(* CODESYS project InstalacaoPortuaria.project

Project tree, tasks and I/O mapping:
  Device : CODESYS Control Win V3, 3S - Smart Software Solutions GmbH, order no. 305021, version 3.5.11.40
    application Application
      libraries: Standard, * (System)
      task MainTask (cyclic, interval t#20ms, priority 0) calls PLC_PRG
      task Simulacao (cyclic, interval t#500ms, priority 1) calls SIMULACAO
      program PLC_PRG [SFC]: _aDESCARREGAMENTO_active, _aCARREGAMENTO_active, _aALARMES_active, _aS5_entry, _aSC2_entry, _aSC3_entry, _aSC4_entry, _aSC5_entry, _aSC6_entry, _aSC7_entry, _aS7_active, _aSC10_active, _aS1_active, _aSC2_active, _aSELECAO_DESC_active, _aSELECAO_CARR_active, _aInit_active, _aS3_active
      program SIMULACAO [SFC]: _aSCARREGAMENTO_active, _aSDESCARREGAMENTO_active, _aSD2_active, _aSD3_entry, _aSC2_active, _aSSILO_active, _aSC3_entry, _aSD1_entry, _aSC0_entry, _aSC0_exit, _aSC3_exit, _aSD0_entry, _aSD0_exit, _aSD3_exit
      Symbols
*)

// Device/Application/PLC_PRG
PROGRAM PLC_PRG
VAR_INPUT
	// VAGAO GRANELEIRO
	// VARIAVEL REFERENTE AO SENSOR DE POSICIONAMENTO DO VAGAO GRANELEIRO
	VAGAO: BOOL:= 0;
	// QUANTIDADE DE GRAOS NO VAGAO GANELEIRO
	GRAOS: REAL:=0;
	
	// TRANSPORTADOR DE ENTRADA
	// CELULA DE CARGA DO TRANSPORTADOR
	C_TR_01: BOOL:= 0;
	
	// SILOS DE ARMAZENAGEM
	// CELULAS DE CARGA
	C_AS_01: REAL:= 0;	
	C_AS_02: REAL:= 0;
	// CHAVE DE BAIXO NIVEL
	L_AS_01: BOOL:= 0;
	L_AS_02: BOOL:= 0;
	// CHAVE DE ALTO NIVEL
	H_AS_01: BOOL:= 0;
	H_AS_02: BOOL:= 0;
	
	// ALIMENTADORES DA MOEGA 
	// INDICADOR DE GRAOS
	C_AL_01: BOOL:= 0;
	C_AL_02: BOOL:= 0;
	
	// MOEGA
	// CONTABILIZA O PESO DOS GRAOS TRANSFERIDOS
	C_MO_01: REAL:= 0;
	
	// TRANSPORTADOR DE SAIDA
	// CELULA DE CARGA DO TRANSPORTADOR
	C_TR_02: BOOL:= 0;
	
	// ALIMENTADOR DE SAIDA
	// SENSOR CAMINHAO CORRETAMENTE POSICIONADO
	CAMINHAO: BOOL:= 0;
	
	// SENSORES DE CHEGADA
	// CHEGADA VAGAO
	VAGAO_C: BOOL:= 0;
	// CHEGADA CAMINHAO
	CAMINHAO_C: BOOL:= 0;
	
	// SENSORES DE SAIDA
	// SAIDA VAGAO
	VAGAO_S: BOOL:= 0;
	// SAIDA CAMINHAO
	CAMINHAO_S: BOOL:= 0;

END_VAR
VAR
	// MODO CARREGAMENTO
	SELEC_CARR_MAN: BOOL:= 0;
	CARR_MAN: BOOL:= 0;
	// INICIA CARREGAMENTO AUTOMATICO
	CARREGAR: BOOL:= 0;
	// CARREGAMENTO NÃO PODE SER ACIONADO
	I_NOT_CARR: BOOL:= 0;
	// ALARME GRAOS INSUFICIENTES
	I_GRAOS: BOOL:= 0;
	// MODO DESCARREGAMENTO
	SELEC_DESC_MAN: BOOL:= 0;
	DESC_MAN: BOOL:= 0;
	// DESCARREGAMENTO NÃO PODE SER ACIONADO
	I_NOT_DESC: BOOL:= 0;
	// INICIA DESCARREGAMENTO AUTOMATICO
	DESCARREGAR: BOOL:= 0;		

	// VARIAVEIS DE INTERFACE
	//VAGAO GRANELEIRO
	// SENSOR DE POSICIONAMENTO DO VAGAO GRANELEIRO
	I_VAGAO: BOOL:= 0;
	
	//TRANSPORTADOR DE ENTRADA
	// ESTADO DO TRANSPORTADOR DE ENTRADA
	I_TR_01: BOOL:= 0;
	// CELULA DE CARGA DO TRANSPORTADOR
	I_C_TR_01: BOOL:= 0;
	// INDICACAO QUE O TRANSPORTADOR ESTÁ LIGADO E VAZIO POR MAIS DE 5S
	I_VAZIO_TR_01: BOOL:= 0;
	
	// DESVIADOR DE MANGUEIRA
	I_MG_01: BOOL:= 0;
	
	// SILOS DE ARMAZENAGEM
	// CELULAS DE CARGA
	I_C_AS_01: REAL:= 0;	
	I_C_AS_02: REAL:= 0;
	// CHAVE DE BAIXO NIVEL
	I_L_AS_01: BOOL:= 0;
	I_L_AS_02: BOOL:= 0;
	// CHAVE DE ALTO NIVEL
	I_H_AS_01: BOOL:= 0;
	I_H_AS_02: BOOL:= 0;
	// SISTEMA DE VENTILACAO
	I_V_AS_01: BOOL:= 0;
	I_V_AS_02: BOOL:= 0;
	
	// ALIMENTADORES DA MOEGA 
	I_AL_01: BOOL:= 0;
	I_AL_02: BOOL:= 0;
	// ALARME LIGADO E VAZIO POR MAIS DE 5S
	I_VAZIO_AL_01: BOOL:= 0;
	I_VAZIO_AL_02: BOOL:= 0;
	// INDICADOR DE GRAOS
	I_C_AL_01: BOOL:= 0;
	I_C_AL_02: BOOL:= 0;
	
	// MOEGA
	// ESTADO DA MOEGA
	I_MO_01: BOOL:= 0;
	// CONTABILIZA O PESO DOS GRAOS TRANSFERIDOS
	I_C_MO_01: REAL:= 0;
	// ALARME TRANSPORTADOR DESLIGADO E PESO DIFERENTE DE 0
	I_CHEIO_MO_01: BOOL:= 0; 
	
	//TRANSPORTADOR DE SAIDA
	// ESTADO DO TRANSPORTADOR DE SAIDA
	I_TR_02: BOOL:= 0;
	// CELULA DE CARGA DO TRANSPORTADOR
	I_C_TR_02: BOOL:= 0;
	// INDICACAO QUE O TRANSPORTADOR ESTÁ LIGADO E VAZIO POR MAIS DE 5S
	I_VAZIO_TR_02: BOOL:= 0;
	// INDICACAO QUE O TRANSPORTADOR ESTÁ LIGADO E ALIMENTADOR DESLIGADO
	I_LIGADO_TR_02: BOOL:= 0;
	
	// ALIMENTADOR DE SAIDA
	// ESTADO DO ALIMENTADOR DE SAIDA
	I_AL_03: BOOL:= 0;
	// SENSOR CAMINHAO CORRETAMENTE POSICIONADO
	I_CAMIHAO: BOOL:= 0;
	// ALARME ALIMENTADOR LIGADO CAMINHAO DESCONECTADO
	I_LIGADO_AL_03: BOOL:=0;
	
	// CAPACIDADE DO CAMINHAO
	I_CAPACIDADE: REAL:= 0;
	
	// SENSORES DE CHEGADA
	// CHEGADA VAGAO
	I_VAGAO_C: BOOL:= 0;
	// CHEGADA CAMINHAO
	I_CAMINHAO_C: BOOL:= 0;
	
	// SENSORES DE SAIDA
	// SAIDA VAGAO
	I_VAGAO_S: BOOL:= 0;
	// SAIDA CAMINHAO
	I_CAMINHAO_S: BOOL:= 0;
	
	TON_0: TON;
	TON_1: TON;
END_VAR
VAR_OUTPUT
	
	//TRANSPORTADOR DE ENTRADA
	// ACIONA O TRANSPORTADOR DE ENTRADA
	TR_01: BOOL:= 0;

	//DESVIADOR DE MANGUEIRA
	MG_01: BOOL:= 0;

	// SILOS DE ARMAZENAGEM
	// SISTEMA DE VENTILACAO
	V_AS_01: BOOL:= 0;
	V_AS_02: BOOL:= 0;
	
	//ALIMENTADORES DA MOEGA 
	AL_01: BOOL:= 0;
	AL_02: BOOL:= 0;
	
	// MOEGA
	// ESTADO DA MOEGA
	MO_01: BOOL:= 0;
	
	//TRANSPORTADOR DE SAIDA
	// ESTADO DO TRANSPORTADOR DE SAIDA
	TR_02: BOOL:= 0;
	
	// ALIMENTADOR DE SAIDA
	// ESTADO DO ALIMENTADOR DE SAIDA
	AL_03: BOOL:= 0;

END_VAR

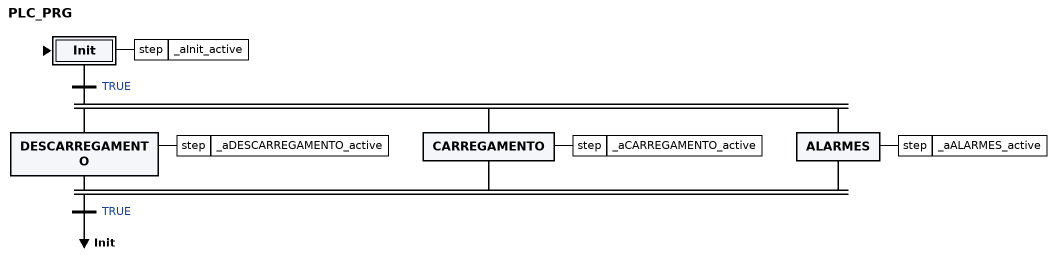
INITIAL_STEP Init:
    _aInit_active(N);  // step action
END_STEP
TRANSITION FROM Init TO (DESCARREGAMENTO, CARREGAMENTO, ALARMES)
    := TRUE;
END_TRANSITION
STEP DESCARREGAMENTO:
    _aDESCARREGAMENTO_active(N);  // step action
END_STEP
STEP CARREGAMENTO:
    _aCARREGAMENTO_active(N);  // step action
END_STEP
STEP ALARMES:
    _aALARMES_active(N);  // step action
END_STEP
TRANSITION FROM (DESCARREGAMENTO, CARREGAMENTO, ALARMES) TO Init
    := TRUE;
END_TRANSITION

ACTION _aDESCARREGAMENTO_active:
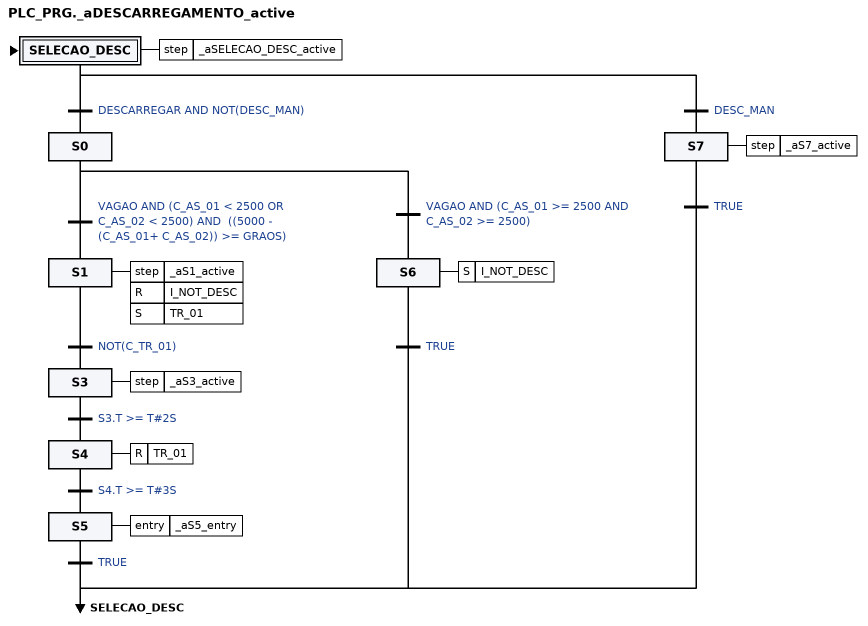
INITIAL_STEP SELECAO_DESC:
    _aSELECAO_DESC_active(N);  // step action
END_STEP
TRANSITION FROM SELECAO_DESC TO S0
    := DESCARREGAR AND NOT(DESC_MAN);
END_TRANSITION
STEP S0:
END_STEP
TRANSITION FROM S0 TO S1
    := VAGAO AND (C_AS_01 < 2500 OR C_AS_02 < 2500) AND ((5000 - (C_AS_01+ C_AS_02)) >= GRAOS);
END_TRANSITION
STEP S1:
    _aS1_active(N);  // step action
    I_NOT_DESC(R);
    TR_01(S);
END_STEP
TRANSITION FROM S1 TO S3
    := NOT(C_TR_01);
END_TRANSITION
STEP S3:
    _aS3_active(N);  // step action
END_STEP
TRANSITION FROM S3 TO S4
    := S3.T >= T#2S;
END_TRANSITION
STEP S4:
    TR_01(R);
END_STEP
TRANSITION FROM S4 TO S5
    := S4.T >= T#3S;
END_TRANSITION
STEP S5:
    _aS5_entry(P1);  // entry action
END_STEP
TRANSITION FROM S5 TO SELECAO_DESC
    := TRUE;
END_TRANSITION
TRANSITION FROM S0 TO S6
    := VAGAO AND (C_AS_01 >= 2500 AND C_AS_02 >= 2500);
END_TRANSITION
STEP S6:
    I_NOT_DESC(S);
END_STEP
TRANSITION FROM S6 TO SELECAO_DESC
    := TRUE;
END_TRANSITION
TRANSITION FROM SELECAO_DESC TO S7
    := DESC_MAN;
END_TRANSITION
STEP S7:
    _aS7_active(N);  // step action
END_STEP
TRANSITION FROM S7 TO SELECAO_DESC
    := TRUE;
END_TRANSITION
// branch label Branch2__aDESCARREGAMENTO_entry
END_ACTION

ACTION _aCARREGAMENTO_active:
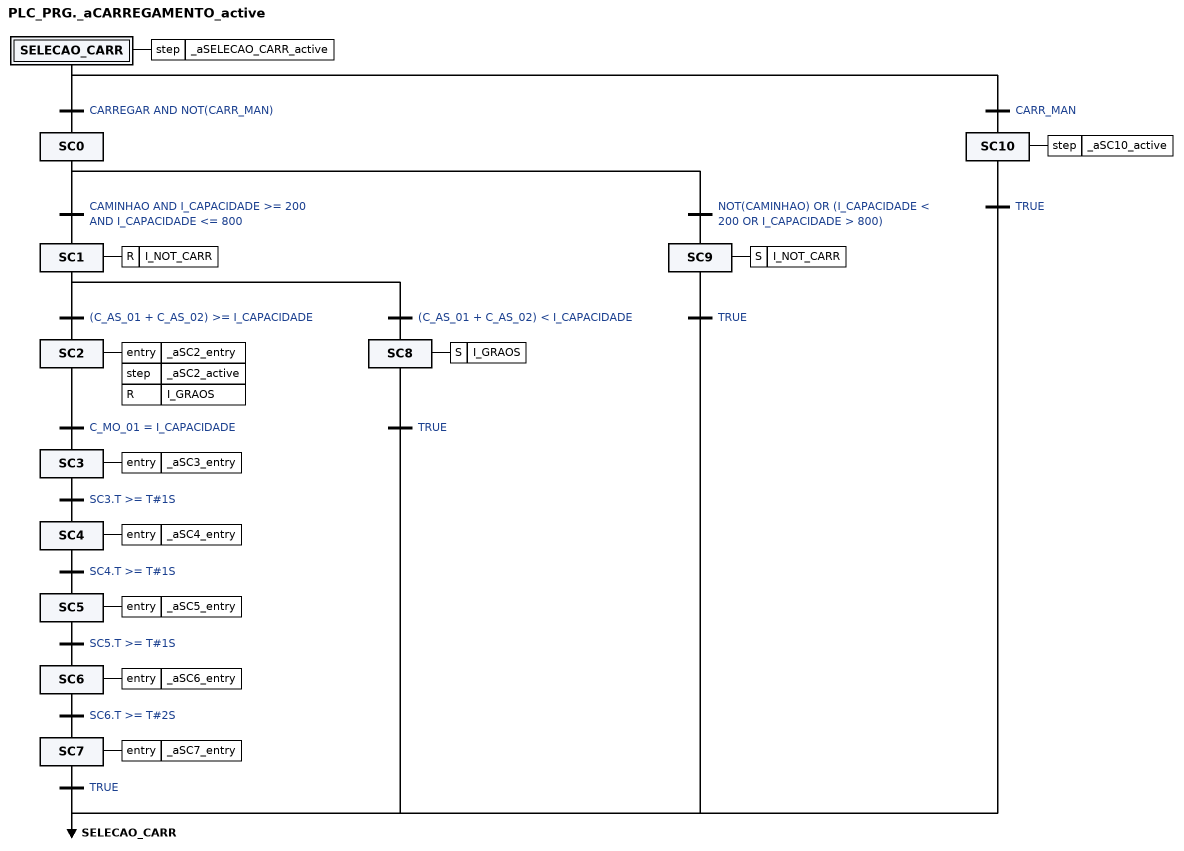
INITIAL_STEP _SELECAO_CARR:  // name as stored:  SELECAO_CARR
    _aSELECAO_CARR_active(N);  // step action
END_STEP
TRANSITION FROM _SELECAO_CARR TO SC0
    := CARREGAR AND NOT(CARR_MAN);
END_TRANSITION
STEP SC0:
END_STEP
TRANSITION FROM SC0 TO SC1
    := CAMINHAO AND I_CAPACIDADE >= 200 AND I_CAPACIDADE <= 800;
END_TRANSITION
STEP SC1:
    I_NOT_CARR(R);
END_STEP
TRANSITION FROM SC1 TO SC2
    := (C_AS_01 + C_AS_02) >= I_CAPACIDADE;
END_TRANSITION
STEP SC2:
    _aSC2_entry(P1);  // entry action
    _aSC2_active(N);  // step action
    I_GRAOS(R);
END_STEP
TRANSITION FROM SC2 TO SC3
    := C_MO_01 = I_CAPACIDADE;
END_TRANSITION
STEP SC3:
    _aSC3_entry(P1);  // entry action
END_STEP
TRANSITION FROM SC3 TO SC4
    := SC3.T >= T#1S;
END_TRANSITION
STEP SC4:
    _aSC4_entry(P1);  // entry action
END_STEP
TRANSITION FROM SC4 TO SC5
    := SC4.T >= T#1S;
END_TRANSITION
STEP SC5:
    _aSC5_entry(P1);  // entry action
END_STEP
TRANSITION FROM SC5 TO SC6
    := SC5.T >= T#1S;
END_TRANSITION
STEP SC6:
    _aSC6_entry(P1);  // entry action
END_STEP
TRANSITION FROM SC6 TO SC7
    := SC6.T >= T#2S;
END_TRANSITION
STEP SC7:
    _aSC7_entry(P1);  // entry action
END_STEP
TRANSITION FROM SC7 TO SELECAO_CARR
    := TRUE;
END_TRANSITION
TRANSITION FROM SC1 TO SC8
    := (C_AS_01 + C_AS_02) < I_CAPACIDADE;
END_TRANSITION
STEP SC8:
    I_GRAOS(S);
END_STEP
TRANSITION FROM SC8 TO SELECAO_CARR
    := TRUE;
END_TRANSITION
TRANSITION FROM SC0 TO SC9
    := NOT(CAMINHAO) OR (I_CAPACIDADE < 200 OR I_CAPACIDADE > 800);
END_TRANSITION
STEP SC9:
    I_NOT_CARR(S);
END_STEP
TRANSITION FROM SC9 TO SELECAO_CARR
    := TRUE;
END_TRANSITION
TRANSITION FROM _SELECAO_CARR TO SC10
    := CARR_MAN;
END_TRANSITION
STEP SC10:
    _aSC10_active(N);  // step action
END_STEP
TRANSITION FROM SC10 TO SELECAO_CARR
    := TRUE;
END_TRANSITION
// branch label Branch2__aCARREGAMENTO_active
// branch label Branch1__aCARREGAMENTO_active
// branch label Branch0__aCARREGAMENTO_active
END_ACTION

ACTION _aALARMES_active:
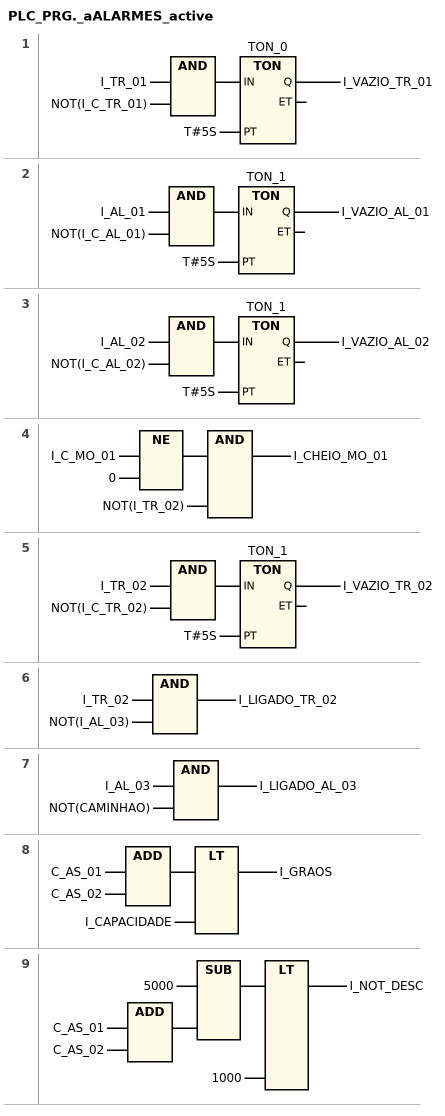
// NETWORK 1
TON_0(IN := I_TR_01 AND (NOT(I_C_TR_01)), PT := T#5S); // TON
I_VAZIO_TR_01 := TON_0.Q;

// NETWORK 2
TON_1(IN := I_AL_01 AND (NOT(I_C_AL_01)), PT := T#5S); // TON
I_VAZIO_AL_01 := TON_1.Q;

// NETWORK 3
TON_1(IN := I_AL_02 AND (NOT(I_C_AL_02)), PT := T#5S); // TON
I_VAZIO_AL_02 := TON_1.Q;

// NETWORK 4
I_CHEIO_MO_01 := I_C_MO_01 <> 0 AND (NOT(I_TR_02));

// NETWORK 5
TON_1(IN := I_TR_02 AND (NOT(I_C_TR_02)), PT := T#5S); // TON
I_VAZIO_TR_02 := TON_1.Q;

// NETWORK 6
I_LIGADO_TR_02 := I_TR_02 AND (NOT(I_AL_03));

// NETWORK 7
I_LIGADO_AL_03 := I_AL_03 AND (NOT(CAMINHAO));

// NETWORK 8
I_GRAOS := C_AS_01 + C_AS_02 < I_CAPACIDADE;

// NETWORK 9
I_NOT_DESC := 5000 - (C_AS_01 + C_AS_02) < 1000;
END_ACTION

ACTION _aS5_entry:
IF (I_V_AS_01 = 1) THEN
	V_AS_01:= 0;
END_IF
IF (I_V_AS_02 = 1) THEN
	V_AS_02:= 0;
END_IF
I_V_AS_01:= V_AS_01;
I_V_AS_02:= V_AS_02;
END_ACTION

ACTION _aSC2_entry:
//ALIMENTADOR DE SAÍDA
AL_03 := 1;
I_AL_03 := AL_03;
//TRANSPORTADOR DE SAÍDA
TR_02 := 1;
I_TR_02 := TR_02;
//MOEGA
MO_01 := 1;
I_MO_01 := MO_01;
END_ACTION

ACTION _aSC3_entry:
//SILO
IF (I_AL_01 = 1) THEN
	AL_01 := 0;
END_IF
IF (I_AL_02 = 1) THEN
	AL_02 := 0;
END_IF
I_AL_01 := AL_01;
I_AL_02 := AL_02;
END_ACTION

ACTION _aSC4_entry:
//MOEGA
MO_01 := 0;
I_MO_01 := MO_01;
END_ACTION

ACTION _aSC5_entry:
//TRANSPORTADOR DE SAÍDA
TR_02 := 0;
I_TR_02 := TR_02;
END_ACTION

ACTION _aSC6_entry:
//ALIMENTADOR DE SAÍDA
AL_03 := 0;
I_AL_03 := AL_03;
END_ACTION

ACTION _aSC7_entry:
//SILO
IF (I_V_AS_01 = 1) THEN
	V_AS_01 := 0;
END_IF
IF (I_V_AS_02 = 1) THEN
	V_AS_02 := 0;
END_IF
I_V_AS_01 := V_AS_01;
I_V_AS_02 := V_AS_02;
END_ACTION

ACTION _aS7_active:
// TRANSPORTADOR DE ENTRADA
IF(I_TR_01 = 1)THEN
	TR_01:= 1;
ELSE
	TR_01:= 0;
END_IF
// DESVIADOR DA MANGUEIRA
IF(I_MG_01 = 1)THEN
	MG_01:= 1;
ELSE
	MG_01:= 0;
END_IF
// SILO DE ARMAZENAGEM 1
IF(I_V_AS_01 = 1)THEN
	V_AS_01:= 1;
ELSE
	V_AS_01:= 0;
END_IF
// SILO DE ARMAZENAGEM 2
IF(I_V_AS_02 = 1)THEN
	V_AS_02:= 1;
ELSE
	V_AS_02:= 0;
END_IF
END_ACTION

ACTION _aSC10_active:
// SILO DE ARMAZENAGEM 1
IF(I_V_AS_01 = 1)THEN
	V_AS_01:= 1;
ELSE
	V_AS_01:= 0;
END_IF
// SILO DE ARMAZENAGEM 2
IF(I_V_AS_02 = 1)THEN
	V_AS_02:= 1;
ELSE
	V_AS_02:= 0;
END_IF
// ALIMENTADOR DA MOEGA 1
IF(I_AL_01 = 1)THEN
	AL_01:= 1;
ELSE
	AL_01:= 0;
END_IF
// ALIMENTADOR DA MOEGA 2
IF(I_AL_02 = 1)THEN
	AL_02:= 1;
ELSE
	AL_02:= 0;
END_IF
// MOEGA
IF(I_MO_01 = 1)THEN
	MO_01:= 1;
ELSE
	MO_01:= 0;
END_IF
// TRANSPORTADOR DE SAÍDA
IF(I_TR_02 = 1)THEN
	TR_02:= 1;
ELSE
	TR_02:= 0;
END_IF
// ALIMENTADOR DE SAÍDA
IF(I_AL_03 = 1)THEN
	AL_03:= 1;
ELSE
	AL_03:= 0;
END_IF
END_ACTION

ACTION _aS1_active:
IF (C_AS_01 <= C_AS_02) THEN
		MG_01:= 0;
ELSE
		MG_01:= 1;
END_IF
I_MG_01:= MG_01;
I_C_AS_01:= C_AS_01; 
I_C_AS_02:= C_AS_02;

IF (I_MG_01 = 0) THEN
	V_AS_01:= 1;
ELSE
	V_AS_02:= 1;
END_IF
I_V_AS_01:= V_AS_01;
I_V_AS_02:= V_AS_02;
END_ACTION

ACTION _aSC2_active:
//SILO
IF (C_AS_01 >= C_AS_02) THEN
		AL_01 := 1;
		AL_02 := 0;
		V_AS_01 := 1;
		V_AS_02 := 0;
ELSE
		AL_01 := 0;
		AL_02 := 1;
		V_AS_01 := 0;
		V_AS_02 := 1;
END_IF
I_AL_01 := AL_01;
I_AL_02 := AL_02;
I_V_AS_01 := V_AS_01;
I_V_AS_02 := V_AS_02;

I_C_AS_01:= C_AS_01; 
I_C_AS_02:= C_AS_02;
END_ACTION

ACTION _aSELECAO_DESC_active:
IF (TR_01 = 0) AND (I_VAZIO_TR_01 = 0) THEN
	DESC_MAN:= SELEC_DESC_MAN;
END_IF
END_ACTION

ACTION _aSELECAO_CARR_active:
IF (AL_01 = 0) AND (AL_02 = 0) AND (AL_03 = 0) AND (MO_01 = 0) AND (TR_02 = 0) 
AND (I_VAZIO_AL_01 = 0) AND (I_VAZIO_AL_02 = 0) AND (I_CHEIO_MO_01 = 0) 
AND (I_VAZIO_TR_02 = 0) AND (I_LIGADO_TR_02 = 0) AND (I_LIGADO_AL_03 = 0)
AND (I_GRAOS = 0) THEN
	CARR_MAN:= SELEC_CARR_MAN;
END_IF
END_ACTION

ACTION _aInit_active:
//CHAVES DE BAIXO NÍVEL
I_L_AS_01:= L_AS_01;
I_L_AS_02:= L_AS_02;
//CHAVES DE ALTO NÍVEL
I_H_AS_01:= H_AS_01;
I_H_AS_02:= H_AS_02;
//SENSORES DE CHEGADA
I_CAMINHAO_C:= CAMINHAO_C;
I_VAGAO_C:= VAGAO_C;
//SENSORES DE SAIDA
I_CAMINHAO_S:= CAMINHAO_S;
I_VAGAO_S:= VAGAO_S;
//SENSOR VAGAO POSICIONADO
I_VAGAO:= VAGAO;
END_ACTION

ACTION _aS3_active:
I_C_AS_01:= C_AS_01; 
I_C_AS_02:= C_AS_02;
END_ACTION

END_PROGRAM

// Device/Application/SIMULACAO
PROGRAM SIMULACAO

VAR
	T1: TON;
	T2: TON;
	GRAOS_VAGAO: REAL := 0;
END_VAR

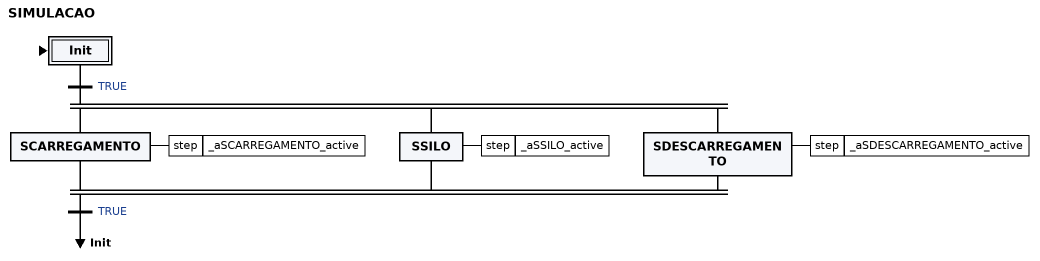
INITIAL_STEP Init:
END_STEP
TRANSITION FROM Init TO (SCARREGAMENTO, SSILO, SDESCARREGAMENTO)
    := TRUE;
END_TRANSITION
STEP SCARREGAMENTO:
    _aSCARREGAMENTO_active(N);  // step action
END_STEP
STEP SSILO:
    _aSSILO_active(N);  // step action
END_STEP
STEP SDESCARREGAMENTO:
    _aSDESCARREGAMENTO_active(N);  // step action
END_STEP
TRANSITION FROM (SCARREGAMENTO, SSILO, SDESCARREGAMENTO) TO Init
    := TRUE;
END_TRANSITION

ACTION _aSCARREGAMENTO_active:
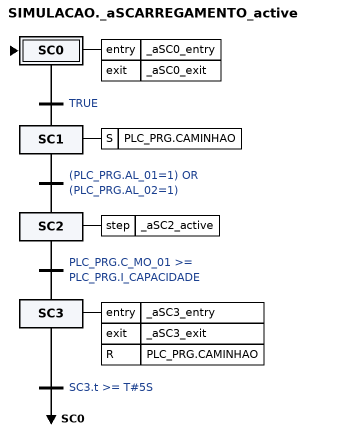
INITIAL_STEP SC0:
    _aSC0_entry(P1);  // entry action
    _aSC0_exit(P0);  // exit action
END_STEP
TRANSITION FROM SC0 TO SC1
    := TRUE;
END_TRANSITION
STEP SC1:
    PLC_PRG.CAMINHAO(S);
END_STEP
TRANSITION FROM SC1 TO SC2
    := (PLC_PRG.AL_01=1) OR (PLC_PRG.AL_02=1);
END_TRANSITION
STEP SC2:
    _aSC2_active(N);  // step action
END_STEP
TRANSITION FROM SC2 TO SC3
    := PLC_PRG.C_MO_01 >= PLC_PRG.I_CAPACIDADE;
END_TRANSITION
STEP SC3:
    _aSC3_entry(P1);  // entry action
    _aSC3_exit(P0);  // exit action
    PLC_PRG.CAMINHAO(R);
END_STEP
TRANSITION FROM SC3 TO SC0
    := SC3.t >= T#5S;
END_TRANSITION
END_ACTION

ACTION _aSDESCARREGAMENTO_active:
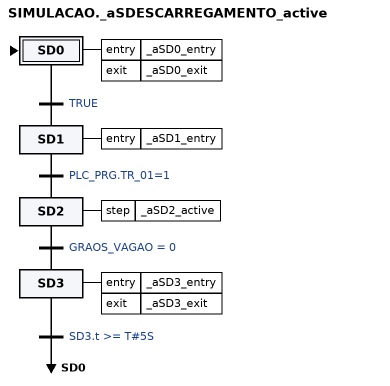
INITIAL_STEP SD0:
    _aSD0_entry(P1);  // entry action
    _aSD0_exit(P0);  // exit action
END_STEP
TRANSITION FROM SD0 TO SD1
    := TRUE;
END_TRANSITION
STEP SD1:
    _aSD1_entry(P1);  // entry action
END_STEP
TRANSITION FROM SD1 TO SD2
    := PLC_PRG.TR_01=1;
END_TRANSITION
STEP SD2:
    _aSD2_active(N);  // step action
END_STEP
TRANSITION FROM SD2 TO SD3
    := GRAOS_VAGAO = 0;
END_TRANSITION
STEP SD3:
    _aSD3_entry(P1);  // entry action
    _aSD3_exit(P0);  // exit action
END_STEP
TRANSITION FROM SD3 TO SD0
    := SD3.t >= T#5S;
END_TRANSITION
END_ACTION

ACTION _aSD2_active:
PLC_PRG.C_TR_01:= 1;
T1(IN:=TRUE,PT:=T#1S);
IF(T1.Q = 1)THEN
	IF (PLC_PRG.MG_01 = 0) THEN
		GRAOS_VAGAO:= GRAOS_VAGAO - 100;
		PLC_PRG.GRAOS:= GRAOS_VAGAO;
		PLC_PRG.C_AS_01:= PLC_PRG.C_AS_01+100;
	ELSE
		GRAOS_VAGAO:= GRAOS_VAGAO - 100;
		PLC_PRG.GRAOS:= GRAOS_VAGAO;
		PLC_PRG.C_AS_02:= PLC_PRG.C_AS_02+100;
	END_IF
	T1(IN:=FALSE);
END_IF
END_ACTION

ACTION _aSD3_entry:
PLC_PRG.C_TR_01:= 0;
PLC_PRG.VAGAO:= 0;
PLC_PRG.VAGAO_S:= 1;
END_ACTION

ACTION _aSC2_active:
PLC_PRG.C_TR_02:= 1;
T2(IN:=TRUE,PT:=T#1S);
IF(T2.Q = 1)THEN
	IF (PLC_PRG.AL_01 = 1) THEN
		IF (PLC_PRG.C_AS_01>=50) THEN
			PLC_PRG.C_AL_01:= 1;
			PLC_PRG.C_AS_01:= PLC_PRG.C_AS_01 - 50;
			PLC_PRG.C_MO_01:= PLC_PRG.C_MO_01 + 50;
		END_IF
	END_IF
	IF (PLC_PRG.AL_02 = 1) THEN
		IF (PLC_PRG.C_AS_02>=50) THEN
			PLC_PRG.C_AL_02:= 1;
			PLC_PRG.C_AS_02:= PLC_PRG.C_AS_02 - 50;
			PLC_PRG.C_MO_01:= PLC_PRG.C_MO_01 + 50;
		END_IF
	END_IF
	T2(IN:=FALSE);
END_IF
END_ACTION

ACTION _aSSILO_active:
//SIMULAÇÃO DAS CHAVES DE ALTO E BAIXO NÍVEL DOS SILOS

IF (PLC_PRG.C_AS_01<=100) THEN
	PLC_PRG.L_AS_01:= 1;
ELSIF (PLC_PRG.C_AS_01>=2400) THEN
	PLC_PRG.H_AS_01:= 1;
ELSE 
	PLC_PRG.L_AS_01:= 0;
	PLC_PRG.H_AS_01:= 0;
END_IF

IF (PLC_PRG.C_AS_02<=100) THEN
	PLC_PRG.L_AS_02:= 1;
ELSIF (PLC_PRG.C_AS_02>=2400) THEN
	PLC_PRG.H_AS_02:= 1;
ELSE 
	PLC_PRG.L_AS_02:= 0;
	PLC_PRG.H_AS_02:= 0;
END_IF
END_ACTION

ACTION _aSC3_entry:
PLC_PRG.C_TR_02:= 0;
PLC_PRG.C_AL_01:= 0;
PLC_PRG.C_AL_02:= 0;
PLC_PRG.C_MO_01:= 0;
PLC_PRG.CAMINHAO_S:= 1;
END_ACTION

ACTION _aSD1_entry:
PLC_PRG.VAGAO:= 1;
GRAOS_VAGAO:= 1000;
PLC_PRG.GRAOS:= GRAOS_VAGAO;
END_ACTION

ACTION _aSC0_entry:
PLC_PRG.CAMINHAO_C:= 1;
END_ACTION

ACTION _aSC0_exit:
PLC_PRG.CAMINHAO_C:= 0;
END_ACTION

ACTION _aSC3_exit:
PLC_PRG.CAMINHAO_S:= 0;
END_ACTION

ACTION _aSD0_entry:
PLC_PRG.VAGAO_C:= 1;
END_ACTION

ACTION _aSD0_exit:
PLC_PRG.VAGAO_C:= 0;
END_ACTION

ACTION _aSD3_exit:
PLC_PRG.VAGAO_S:= 0;
END_ACTION

END_PROGRAM
